Staubli VAL3: F2_gohome.pgx

program F2_gohome()
  local joint l_jTemp1
  local bool l_bTemp
begin
  popUpMsg("ok")
  // go to pfrmCad[1] position
  if size(pfrmCad)>1
    //            //movej(jHome,tTool,mSlow)
    //            movej(jCad[1],flange,mSlow)
    MoveTo.trsf=pfrmCad[0].trsf
    l_bTemp=pointToJoint(tTool,jConfig,MoveTo,l_jTemp1)
    //    $movejSync(jJointRx[l_nCount])
    l_jTemp1.j6=0
    movej(l_jTemp1,tTool,mNomSpeed)
    waitEndMove()
  else
    popUpMsg("Motion need be initilized")
  endIf
end
